FUNCTION_BLOCK FB_FoodWeightModule
VAR_INPUT
	nLine					: INT;
	UnitID					: BYTE;
	fFast_Speed				: REAL;
	fSlow_Speed_1			: REAL;
	fSlow_Speed_2			: REAL;
	fDerisedWeight_Food		: REAL;
	fChangeMode_Food_1		: REAL;
	fChangeMode_Food_2		: REAL;
	fMaxWeight_Food			: REAL;
	fPerStop_Food			: REAL;
	fTimer_Food				: REAL;
	fTimer_Alarm_Food		: REAL;
	fTimer_Check_Food		: REAL;
	fTimer_Error_Food		: REAL;
	fDelta_Food				: REAL;
	fTimer_Reverse			: REAL;
END_VAR
VAR_OUTPUT
	fProductLogF			: ARRAY [1..5] OF REAL;
	bStatus_Food			: BOOL;
	Time_start				: DT;
	Time_Stop				: DT;
	status					: STRING;
	fweight_iot				: REAL;
END_VAR
VAR
	// ===== CHILD COMPONENTS ============
	fbDriver			: FB_Inverter;
	fbLoadcell			: FB_Loadcell;
	// ===== SIM COMPONENTS ==============
	fbDriverSim			: FB_Inverter_Sim;
	fbLoadcellSim		: FB_LoadCell_Sim;
	// ===== INTERFACES ==================
	iDriver				: I_Inverter;
	iLoadcell			: I_LoadCell;
	// ====== VAR IO =====================
	bCupPresent 	AT %I*	: BOOL;
	bError_Driver   AT %I* 	: BOOL;
	//======= VAR METHOD =================
	nState				: INT;
	nStateErr			: INT;
	nStateWrn			: INT;
	fbTimer				: TON;
	fbTimer1			: TON;
	fbTimer_Alarm		: TON;
	fbTimer_Error		: TON;			
	fFastWeight			: REAL;
	fSlowWeight			: REAL;
	fSlowWeight1		: REAL;
	fChangemode_val		: REAL;
	fChangemode_val1	: REAL;
	fLowToleWeight		: REAL;
	fHighToleWeight		: REAL;
	fTareWeight			: REAL;
	bDone				: BOOL;
	p,k					: INT;
	//========= VAR HMI Worm Weight Auto ============
	fFlow_Food						: REAL;
	fWeight_Food					: REAL;
	fActDelta_Food					: REAL;	
	fSpeed_Food_Motor_Manual		: REAL;
	fTime							: REAL;
	Error							: BOOL;
	bStatus							: BOOL;
	timestart						: dt;
END_VAR

IF bSimMode THEN
	iDriver	:= fbDriverSim;
	fbDriverSim();
	iLoadcell	:= fbLoadcellSim;
	fbLoadcellSim();
ELSE
	iDriver	:= fbDriver;
	fbDriver(UnitID := UnitID, id := 2);
	iLoadcell	:= fbLoadcell;
	fbLoadcell(idDevice := nLine,Error => Error);
END_IF

IF iLoadcell.fActWeight > fMaxWeight_Food THEN
	IF nLine = 1 THEN
		F_SetError(56,nLine := 1);
	ELSIF nLine = 2 THEN
		F_SetError(58,nLine := 2);
	END_IF
END_IF

IF Error THEN
	IF nLine = 1 THEN
		F_SetError(69,nLine := 1);
	ELSIF nLine = 2 THEN
		F_SetError(71,nLine := 2);
	END_IF
END_IF

IF bIsError_Driver THEN
	iDriver.Stop();
	IF nLine = 1 THEN
		F_SetError(7,nLine := 1);
	ELSIF nLine = 2 THEN
		F_SetError(29,nLine := 2);
	END_IF
END_IF

METHOD Auto : BOOL
VAR_INPUT
END_VAR

VAR
END_VAR
GetLocalSystemTime(bEnable := 1);
fbTimer(PT := T#100S);
fbTimer_Alarm(PT := REAL_TO_TIME(fTimer_Alarm_Food)*1000);
CASE nState OF
	0:// Init Value
		Auto					:= FALSE;
		fbTimer(IN := FALSE);
		fbTimer1(IN := FALSE);
		fbTimer_Alarm(IN := FALSE);
		fbTimer_Error(IN := FALSE);
		bDone					:= FALSE;
		iDriver.fTargetSpeed 	:= fFast_Speed;
		nState 					:= 1;
	1:// Init Value
		fFastWeight				:= fFast_Speed;
		fSlowWeight				:= fSlow_Speed_1;
		fSlowWeight1			:= fSlow_Speed_2;
		fChangemode_val			:= fDerisedWeight_Food*fChangeMode_Food_1/100;
		fChangemode_val1		:= (fDerisedWeight_Food - fChangemode_val)*fChangeMode_Food_2/100 + fChangemode_val;
		fLowToleWeight			:= fDerisedWeight_Food*(1-(fDelta_Food/100));
		fHighToleWeight			:= fDerisedWeight_Food*(1+(fDelta_Food/100));
		bStatus_Food			:= FALSE;
		bStatus					:= FALSE;
		fTime					:= 0;
		nState					:= 2;
	2:// Cup detection
		iDriver.fTargetSpeed 	:= fFastWeight;
		iLoadcell.NetMode();
		IF NOT bIsCupPresent THEN
			fbTimer1(IN := TRUE, PT := REAL_TO_TIME(fTimer_Food)*1000);
			IF fbTimer1.Q THEN
				nState	:= 3;
			END_IF
		END_IF
	3:// Tare weight
		timestart := SYSTEMTIME_TO_DT(GetLocalSystemTime.systemTime);
		fbTimer1(IN := FALSE);
		fTareWeight 			:= iLoadcell.fActWeight;
		fWeight_Food			:= iLoadcell.fActWeight - fTareWeight;
		nState					:= 4;
	4:
		iDriver.Start();
		iDriver.fTargetSpeed	:= fSlowWeight;
		fbTimer_Alarm(IN := TRUE);
		fTime := TIME_TO_REAL(fbTimer.ET)/1000;
		fWeight_Food			:= iLoadcell.fActWeight - fTareWeight;
		fbTimer(IN := TRUE);
		fFlow_Food				:= fWeight_Food/((TIME_TO_REAL(fbTimer.ET)+0.00001)/1000);
		IF fWeight_Food >= fChangemode_val THEN
			nState 				:= 5;
		END_IF
	5:// Slow 1 Weight
		iDriver.Stop();
		nState					:= 55;
	55:
		iDriver.Start();
		iDriver.fTargetSpeed	:= fSlowWeight;
		fWeight_Food			:= iLoadcell.fActWeight	- fTareWeight;
		fbTimer(IN := TRUE);
		fTime := TIME_TO_REAL(fbTimer.ET)/1000;
		fFlow_Food				:= fWeight_Food/((TIME_TO_REAL(fbTimer.ET)+0.00001)/1000);
		IF fWeight_Food	>= fChangemode_val1 THEN
			nState				:= 6;
		END_IF
	6:// Slow 2 Weight
		iDriver.Stop();
		nState					:= 66;
	66:
		iDriver.fTargetSpeed	:= fSlowWeight1;
		iDriver.Start();
		fWeight_Food			:= iLoadcell.fActWeight	- fTareWeight;
		fbTimer(IN := TRUE);
		fTime := TIME_TO_REAL(fbTimer.ET)/1000;
		fFlow_Food				:= fWeight_Food/((TIME_TO_REAL(fbTimer.ET)+0.00001)/1000);
		IF fWeight_Food	>= fLowToleWeight*fPerStop_Food/100 THEN
			nState				:= 7;
		END_IF
	7:
		iDriver.Stop();
		nState					:= 71;
	71:
		iDriver.Reverse();
		fbTimer(IN := TRUE);
		fWeight_Food			:= iLoadcell.fActWeight	- fTareWeight;
		fbTimer1(IN := TRUE, PT := REAL_TO_TIME(fTimer_Reverse)*1000);
		fTime := TIME_TO_REAL(fbTimer.ET)/1000;
		IF fbTimer1.Q THEN
			nState 				:= 72;
		END_IF
	72:
		fbTimer1(IN := FALSE);
			nState				:= 73;
	73:// Wait Stable Weight
		iDriver.fTargetSpeed 	:= fFastWeight;
		iDriver.Stop();
		fTime := TIME_TO_REAL(fbTimer.ET)/1000;
		fbTimer(IN := TRUE);
		fWeight_Food			:= iLoadcell.fActWeight	- fTareWeight;
		fbTimer1(IN := TRUE, PT := REAL_TO_TIME(fTimer_Check_Food)*1000);
		IF fbTimer1.Q THEN
			nState				:= 8;
		END_IF
	8:// Check Done
		fbTimer1(IN := FALSE);
		fbTimer_Alarm(IN := TRUE);
		fWeight_Food			:= iLoadcell.fActWeight	- fTareWeight;
		IF fWeight_Food < fLowToleWeight THEN
			nState				:= 9;
		ELSIF fWeight_Food >= fLowToleWeight AND fWeight_Food <= fHighToleWeight THEN
			nState				:= 10;
		ELSIF fWeight_Food > fHighToleWeight THEN
			nState				:= 11;	
		END_IF
	9:// No Enough Weight
		fWeight_Food			:= iLoadcell.fActWeight - fTareWeight;
		iDriver.fTargetSpeed	:= fSlowWeight1;
		iDriver.Start();
		IF fWeight_Food	>= fLowToleWeight THEN
			nState				:= 7;
		END_IF
	10:// Enough Weight
		fActDelta_Food			:= (fWeight_food - fDerisedWeight_Food)/fDerisedWeight_Food*100;
		fWeight_Food			:= iLoadcell.fActWeight - fTareWeight;
		fweight_iot				:= iLoadcell.fActWeight - fTareWeight;
		Time_start				:= timestart;
		bStatus_Food			:= TRUE;
		status					:= 'Pass';
		fbTimer(IN := FALSE);
		fbTimer_Alarm(IN := FALSE);
		bDone					:= TRUE;
		p						:= p + 1;
		nState					:= 12;
	11:// Overweight
		fActDelta_Food			:= (fWeight_Food - fDerisedWeight_Food)/fDerisedWeight_Food*100;
		fWeight_Food			:= iLoadcell.fActWeight - fTareWeight;
		fweight_iot				:= iLoadcell.fActWeight - fTareWeight;
		Time_start				:= timestart;
		bStatus_Food			:= FALSE;
		status					:= 'Fail';
		fbTimer_Alarm(IN := FALSE);
		fbTimer(IN := FALSE);
		fbTimer_Error(IN := FALSE);
		bDone					:= TRUE;
		p						:= p + 1;
		IF nLine = 1 THEN
			//F_SetWarning(104);
			nState				:= 12;
		ELSIF nLine = 2 THEN
			//F_SetWarning(111);
			nState				:= 12;
		END_IF
	12:// Done
		Time_Stop				:= SYSTEMTIME_TO_DT(GetLocalSystemTime.systemTime);
		bStatus					:= TRUE;
		IF p > 5 THEN
			p := 5;
		END_IF
		IF bDone THEN
			IF p <> 1 THEN
				FOR k := p TO 2 BY -1 DO
					fProductLogF[k] := fProductLogF[k-1];
				END_FOR
			END_IF
			fProductLogF[1]	:= fWeight_Food;
			bDone 			:= FALSE;
		END_IF
		Auto					:= TRUE;
		nState					:= 13;
	13:
		nState					:= 0;
END_CASE

//Check Timer WormWeight
CASE nStateWrn OF 
	0:
		IF fbTimer_Alarm.Q THEN
			IF nLine = 1 THEN
				F_SetWarning(103,nLine := 1);
			ELSIF nLine = 2 THEN
				F_SetWarning(110,nLine := 2);
			END_IF
			nStateWrn := 1;
		END_IF
	1:
		IF NOT fbTimer_Alarm.Q THEN
			IF nLine = 1 THEN
				bWrn := FALSE;
			ELSIF nLine = 2 THEN
				bWrn2 := FALSE;
			END_IF
			bSirens := FALSE;
			nStateWrn := 0;
		END_IF
		fbTimer_Error(IN := TRUE, PT := REAL_TO_TIME(fTimer_Error_Food*1000));
		IF fbTimer_Error.Q THEN
			IF nLine = 1 THEN
				F_SetError(76,nLine := 1);
			ELSIF nLine = 2 THEN
				F_SetError(78,nLine := 2);
			END_IF
			fbTimer_Alarm(IN := FALSE);
			nState := 11;
			nStateWrn := 0;
		END_IF	
END_CASE

// Check Fault CupPresent

IF nState > 2 AND nState < 99 THEN
	IF bIsCupPresent THEN
		IF nLine = 1 THEN
			F_SetError(45,nLine := 1);
			nState := 0;
		ELSIF nLine = 2 THEN
			F_SetError(46,nLine := 2);
			nState := 0;
		END_IF
	END_IF
END_IF

// Write ProductLog
END_METHOD

PROPERTY bIsCupPresent : BOOL
GET
bIsCupPresent := bCupPresent;
END_GET
END_PROPERTY

PROPERTY bIsError_Driver : BOOL
GET
bIsError_Driver	:= bError_Driver;
END_GET
END_PROPERTY

METHOD Enable : BOOL
VAR_INPUT
END_VAR
iLoadcell.NetMode();
END_METHOD

METHOD Init : BOOL
VAR_INPUT
END_VAR
nState := 0;
END_METHOD

METHOD Manual : BOOL
VAR_INPUT
	bUp_Food_Motor					: BOOL;
	bDown_Food_Motor				: BOOL;
	bZero_Loadcell_Food				: BOOL;
	bMotor_Food						: BOOL;	
	bMotor_Food_Reverse				: BOOL;
END_VAR
IF bUp_Food_Motor THEN
	fSpeed_Food_Motor_Manual	:= fSpeed_Food_Motor_Manual + 10;
END_IF

IF bDown_Food_Motor THEN
	fSpeed_Food_Motor_Manual	:= fSpeed_Food_Motor_Manual - 10;
END_IF

IF bMotor_Food THEN
	iDriver.Start();
ELSIF bMotor_Food_Reverse THEN
	iDriver.Reverse();
ELSIF NOT bMotor_Food AND NOT bMotor_Food_Reverse THEN
	iDriver.Stop();
END_IF

iDriver.fTargetSpeed	:= fSpeed_Food_Motor_Manual;

IF bZero_Loadcell_Food THEN
	iLoadcell.Set_Zero();
ELSE
	iLoadcell.NetMode();
END_IF

fWeight_Food := iLoadcell.fActWeight;
END_METHOD

METHOD Reset : BOOL
VAR_INPUT
END_VAR
iDriver.Reset();
fbTimer(IN := FALSE);			
fbTimer1(IN	:= FALSE);
fbTimer_Alarm(IN := FALSE);
fbTimer_Error(IN := FALSE);
END_METHOD

METHOD SetZero : BOOL
VAR_INPUT
END_VAR
iLoadcell.Set_Zero();
END_METHOD

METHOD Stop : BOOL
VAR_INPUT
END_VAR
iDriver.Stop();
fbTimer(IN := FALSE);			
fbTimer1(IN	:= FALSE);
fbTimer_Alarm(IN := FALSE);
fbTimer_Error(IN := FALSE);
END_METHOD

END_FUNCTION_BLOCK

(* stored: Version 1.1.0.1, ProductVersion 3.1.4024.12
   POU FB_FoodWeightModule: Id {2bac8a86-a7be-46cf-b081-b2bfb82788ea}, SpecialFunc None
   Method Auto: Id {cf3f48ec-bc8a-40e4-a115-502ff292a9f9}
   Property bIsCupPresent: Id {78396d6d-759b-48e9-9927-43cb1e73cecc}
   Get Get: Id {ea48f357-602c-41ec-becb-a66da980d5ee}
   Property bIsError_Driver: Id {619508a9-bc70-4c3a-865d-c1b421677562}
   Get Get: Id {8a96df28-23ae-4d87-b05b-81b5002f3e9d}
   Method Enable: Id {0131f7f6-07bc-4687-a13a-47a67fb92ded}
   Method Init: Id {1029c303-1b74-4a57-b71b-2a5d8297dae0}
   Method Manual: Id {ae727d16-c583-40a0-a740-eb0b3e39a217}
   Method Reset: Id {85cd60bf-9828-407c-9ccf-5595942ff8ad}
   Method SetZero: Id {4f9a0ac8-a930-4264-88ad-e4873072a0bc}
   Method Stop: Id {63d319f9-b480-4610-ae39-36aa3a1e2469} *)
